GLOBALCONSTANTS AID_FA_FILL (* Fill attributes object attribute ids *)
  (* Standard: 61499-1; Description: Copyright (c) 2023 HR Agrartechnik GmbH This program and the accompanying materials are made available under the terms of the Eclipse Public License 2.0 which is available at https://www.eclipse.org/legal/epl-2.0/ SPDX-License-Identifier: EPL-2.0 *)
  (* Version 1.0, 2026-06-20, Franz Höpfinger, HR Agrartechnik GmbH *)
  PACKAGE isobus::UT::Q::const::AID;
  IMPORT eclipse4diac::core::TypeHash;
  VAR_GLOBAL CONSTANT
    FILL_TYPE : USINT := USINT#1; (* 1: AID_FA_FILL_FILL_TYPE - Fills: 0=no fill, 1=fill with line colour, 2=fill with specified colour, 3=fill with pattern. *)
    COLOUR : USINT := USINT#2; (* 2: AID_FA_FILL_COLOUR - Colour index. *)
    PATTERN : USINT := USINT#3; (* 3: AID_FA_FILL_PATTERN *)
  END_VAR
END_GLOBALCONSTANTS
